Yaskawa INFORM job: R1_W12(125,90)(KAMERA).JBI

/JOB
//NAME R1_W12(125,90)(KAMERA)
///FOLDERNAME SCIANA-NOWY-R2-KM
//POS
///NPOS 15,15,0,0,0,0
///TOOL 0
///POSTYPE PULSE
///PULSE
C00000=167342,-92471,-131631,-15300,65044,-71165
C00001=162457,-153227,-130225,463,96631,-68116
C00002=73849,-162743,-118840,3050,77824,6167
C00003=-56151,-123607,-84681,24015,93824,29050
C00004=-38514,-119451,-74638,22450,88065,28099
C00005=-45017,-112529,-69741,24595,90810,25157
C00006=60796,-15342,30656,-25990,89314,-17670
C00007=59751,-12665,34197,-26363,88297,-17792
C00008=-31806,-120206,-72760,27731,85167,28638
C00009=-11756,-120523,-68261,34686,77250,33384
C00010=-16104,-135523,-87595,33683,82412,33282
C00011=-16104,-134772,-86650,33694,82248,33232
C00012=-16104,-134772,-86650,33694,82248,-81437
C00013=-16104,-134772,-86650,33694,31806,-81437
C00014=-17357,-183139,-134392,16915,3390,-73963
BC00000=336449,1346288,1069314
BC00001=317239,1346288,1023433
BC00002=255189,1304147,526431
BC00003=206273,1310433,258838
BC00004=160484,1192669,297430
BC00005=154972,1192689,258838
BC00006=114520,1192678,539252
BC00007=114520,1192678,539252
BC00008=154972,1192689,258838
BC00009=154972,1192689,258838
BC00010=154972,1192689,258838
BC00011=154972,1192689,777183
BC00012=154972,1192689,777183
BC00013=154972,1285979,777183
BC00014=154972,1297036,1037732
//INST
///DATE 2024/07/16 20:07
///ATTR SC,RW
///GROUP1 RB1,BS1
NOP
'r1_W12(125,90)(kamera)
'Path W411
SFTOF
MOVJ C00000 BC00000 VJ=100.00
MOVJ C00001 BC00001 VJ=100.00
MOVJ C00002 BC00002 VJ=100.00
MOVJ C00003 BC00003 VJ=100.00
MOVJ C00004 BC00004 VJ=100.00
MOVJ C00005 BC00005 VJ=15.00
REFP 1 C00006 BC00006
REFP 2 C00007 BC00007
MACRO1 MJ#(0) ARGF6
ARCON
WVON WEV#(14)
MOVL C00008 BC00008 V=10.8
MOVL C00009 BC00009 V=10.8
ARCOF
WVOF
MOVL C00010 BC00010 V=333.3
MOVL C00011 BC00011 V=833.3
MOVJ C00012 BC00012 VJ=100.00
MOVJ C00013 BC00013 VJ=100.00
MOVJ C00014 BC00014 VJ=100.00
'Path W412
SFTOF
'W27-1
END
